{warning 'TODO: Implementation'}
FUNCTION_BLOCK PUBLIC FINAL FB_MessageDescriptor
VAR_INPUT
END_VAR
VAR_OUTPUT
END_VAR
VAR
END_VAR

END_FUNCTION_BLOCK

(* stored: Version 1.1.0.1
   POU FB_MessageDescriptor: Id {d624980b-bcaf-4a88-87ae-f3ccdc9b8a97}, SpecialFunc None *)
